{attribute addProperty BoxType "EL5152-0000-0016"}
{attribute addProperty Id "ENC_Status_compact_Channel_1AT %I*ENC_Status_compact_Channel_F561D5116480ENC_Period_Channel_1AT %I*ENC_Period_Channel_AC51B8A03240ENC_Status_compact_Channel_2AT %I*ENC_Status_compact_Channel_F561D5116480ENC_Period_Channel_2AT %I*ENC_Period_Channel_AC51B8A03240ENC_Control_compact_ChannelAT %Q*ARRAY[0..1] OF ENC_Control_compact_Channel_8FDE73944860WcStateAT %I*WcState_F855686C1620InfoDataAT %I*InfoData_BC63D37F80100"}
{attribute addProperty CRC "1657935673"}
{attribute addProperty SizeInBites "336"}
{attribute addProperty SizeInBytes "42"}
TYPE EL5152_0C847284 :
STRUCT
	{attribute addProperty Name "ENC_Status_compact_Channel_1"}
	ENC_Status_compact_Channel_1 : ENC_Status_compact_Channel_F561D511;
	{attribute addProperty Name "ENC_Period_Channel_1"}
	ENC_Period_Channel_1 : ENC_Period_Channel_AC51B8A0;
	{attribute addProperty Name "ENC_Status_compact_Channel_2"}
	ENC_Status_compact_Channel_2 : ENC_Status_compact_Channel_F561D511;
	{attribute addProperty Name "ENC_Period_Channel_2"}
	ENC_Period_Channel_2 : ENC_Period_Channel_AC51B8A0;
	{attribute addProperty Name "ENC_Control_compact_Channel"}
	ENC_Control_compact_Channel : ARRAY[0..1] OF ENC_Control_compact_Channel_8FDE7394;
	{attribute addProperty Name "WcState"}
	WcState : WcState_F855686C;
	{attribute addProperty Name "InfoData"}
	InfoData : InfoData_BC63D37F;
END_STRUCT
END_TYPE

(* stored: Version 1.2.0.0, ProductVersion 3.1.4024.9
   DUT EL5152_0C847284: Id {2136b908-75df-4610-a975-fe748a6b1f96} *)
